// Mitsubishi GX Works2 project: 機電整合乙級第二題-ST   PLC: FX3U/FX3UC

// task Task_01 (event TRUE, interval 0, priority 31): POU_01

PROGRAM POU_01
VAR
  wProgramStep : INT;
  tdT11 : TON;
  tdT10 : TON;
  rtM0 : R_TRIG;
  rtX17 : R_TRIG;
  tdT7 : TON;
  tdT0 : TON;
  rtX2 : R_TRIG;
  ftX2 : F_TRIG;
  tdT200 : TON;
END_VAR
(* 機電整合乙級術科第二題
   Author: Steven Luo
   Date: 2018/10/25
*)

IF M8000 THEN
	RD3A(TRUE, 0, 21, D10);
	MOV(TRUE, K4X0, K4M160);
	MOV(TRUE, K4Y0, K4M180);
END_IF;

IF NOT tdT11.Q THEN
	tdT10(IN := TRUE, PT := T#100ms);
	IF tdT10.Q THEN
		tdT11(IN := TRUE, PT := T#100ms);
		MOVP(TRUE, D10, D4);
	END_IF;
END_IF;

IF M8002 THEN
	rtM0(_CLK := M0);
	rtX17(_CLK := X17);
	wProgramStep := 0;
END_IF;

IF X7 AND X3 AND X5 AND X12 AND X13 AND NOT Y17 AND NOT Y13 AND X2 AND D110 = 0 THEN
	M0 := TRUE;
END_IF;

IF NOT M144 THEN
	IF M0 THEN
		M142 := TRUE;
		M100 := FALSE;
	ELSE
		D5 := 210;
	END_IF;
END_IF;

IF rtM0.Q OR rtX17.Q THEN
	D5 := 0;
END_IF;

IF M10 THEN
	Y5 := TRUE;
	IF X6 THEN
		Y4 := TRUE;
		IF X4 THEN
			IF wProgramStep = 22 OR wProgramStep = 29 THEN
				Y7 := TRUE;
				tdT7(IN := TRUE, PT := T#500ms);
			END_IF;
			IF wProgramStep = 25 OR wProgramStep = 32 THEN
				Y10 := TRUE;
			END_IF;
		END_IF;
	END_IF;
END_IF;

IF M11 THEN
	Y4 := FALSE;
	IF X3 THEN
		Y6 := TRUE;
	END_IF;
END_IF;

IF M20 THEN
	CMP(TRUE, D100, D110, Y1);
	tdT0(IN := TRUE, PT := T#4s);
END_IF;

IF rtX2.Q OR ftX2.Q THEN
	IF Y1 THEN
		INCP(TRUE, D110);
	END_IF;
	IF Y3 THEN
		DECP(TRUE, D110);
	END_IF;
END_IF;

CASE wProgramStep OF
0:
	IF X17 THEN
		IF M130 THEN
			tdT200(IN := FALSE);
			wProgramStep := 200;
		ELSE
			wProgramStep := 20;
		END_IF;
	END_IF;
20:
	IF M130 THEN
		wProgramStep := 0;
	END_IF;
200:
	OUT(M110, Y0);
	IF X3 AND X5 THEN
		IF M111 THEN
			tdT200(IN := TRUE, PT := T#500ms);
			Y3 := TRUE;
		END_IF;
		IF M112 THEN
(*			tdT200(IN := TRUE, PT := T#500ms);*)
			Y1 := TRUE;
		END_IF;
		IF (*(Y1 OR Y3) AND X2 AND*) tdT200.Q THEN
			D1 := 100;
			IF Y3 THEN
				Y3 := FALSE;
			END_IF;
			IF Y1 THEN
				Y1 := FALSE;
			END_IF;
			tdT200(IN := FALSE);
		END_IF;
	END_IF;
	OUT(M113, Y4);
	OUT(M114, Y5);
	OUT(M115, Y6);
	OUT(M116, Y7);
	OUT(M117, Y10);
	OUT(M118, Y17);
	OUT(M119, Y13);
	OUT(M120, Y14);
	OUT(M121, Y15);
	IF NOT M130 THEN
		wProgramStep := 0;
	END_IF;
END_CASE;
END_PROGRAM
